{attribute 'linkalways'} 
{attribute 'no_explicit_call' := 'This FB is a CLASS and must be accessed using methods or properties'}
{attribute 'enable_dynamic_creation'}
FUNCTION_BLOCK Node_F_VN_DrawRectangle_TcVnRectangle_DINT EXTENDS VisionNode
VAR
    stRectangle : _TcVnRectangle_DINT;
    ipDestImage : _ITcVnImage;
    aColor : _TcVnVector4_LREAL;
    nThickness : _DINT(1);
    hrPrev : _HRESULT(S_OK);
	hresult : _HRESULT(S_OK);
END_VAR

METHOD PUBLIC  Clone : I_Node
VAR
	pNode : POINTER TO Node_F_VN_DrawRectangle_TcVnRectangle_DINT;
END_VAR
pNode := __NEW(Node_F_VN_DrawRectangle_TcVnRectangle_DINT);
Clone := pNode^;
END_METHOD

METHOD FB_init : BOOL
VAR_INPUT
	bInitRetains : BOOL; // if TRUE, the retain variables are initialized (warm start / cold start)
	bInCopyCode : BOOL;  // if TRUE, the instance afterwards gets moved into the copy code (online change)
END_VAR
AddInput('stRectangle', stRectangle);
AddInput('ipDestImage', ipDestImage);
AddInput('aColor', aColor);
AddParameter('nThickness', nThickness);
AddInput('hrPrev', hrPrev);
AddOutput('ipDestImage', ipDestImage);
AddOutput('hresult',hresult);
END_METHOD

METHOD PROTECTED OnExecute
hresult.Value := F_VN_DrawRectangle_TcVnRectangle_DINT(
    stRectangle := stRectangle.Value,
	ipDestImage := ipDestImage.Value,
    aColor := aColor.Value,
    nThickness := nThickness.Value,
	hrPrev:= hrPrev.Value);
END_METHOD

METHOD PUBLIC PreExecutionCheck
VAR_INPUT
	Check : I_PreExecutionChecks;
END_VAR
Check.IsTrue(ipDestImage.IsValid, 'ipDestImage must contain an image');
Check.IsTrue(nThickness.Value <> 0, 'nThickness must be non-zero');
END_METHOD

END_FUNCTION_BLOCK

(* stored: Version 1.1.0.1, ProductVersion 3.1.4024.15
   POU Node_F_VN_DrawRectangle_TcVnRectangle_DINT: Id {58dc579c-8f30-0db9-1243-2c96d67bf7bb}, SpecialFunc None
   Folder Constructor: Id {1c9ed1dc-4483-0307-1cae-f313c2c2bde0}
   Method Clone: Id {354bc9c8-89d7-0a92-1aa3-6d1004fb8c62}
   Method FB_init: Id {1d0a65c9-faf0-0395-2111-7ee6ef1c07cc}
   Method OnExecute: Id {a271965c-0fe5-050e-191b-aead3d503403}
   Method PreExecutionCheck: Id {f3bd2c30-d21d-0450-0f08-2e312e644897} *)
